// SIMATIC S7-200 project (STEP 7-Micro/WIN), CPU 224XP REL 02.01

SYMBOL_TABLE USER1
P0               M0.0
END_SYMBOL_TABLE

ORGANIZATION_BLOCK MAIN:OB1
TITLE=PROGRAM COMMENTS
BEGIN
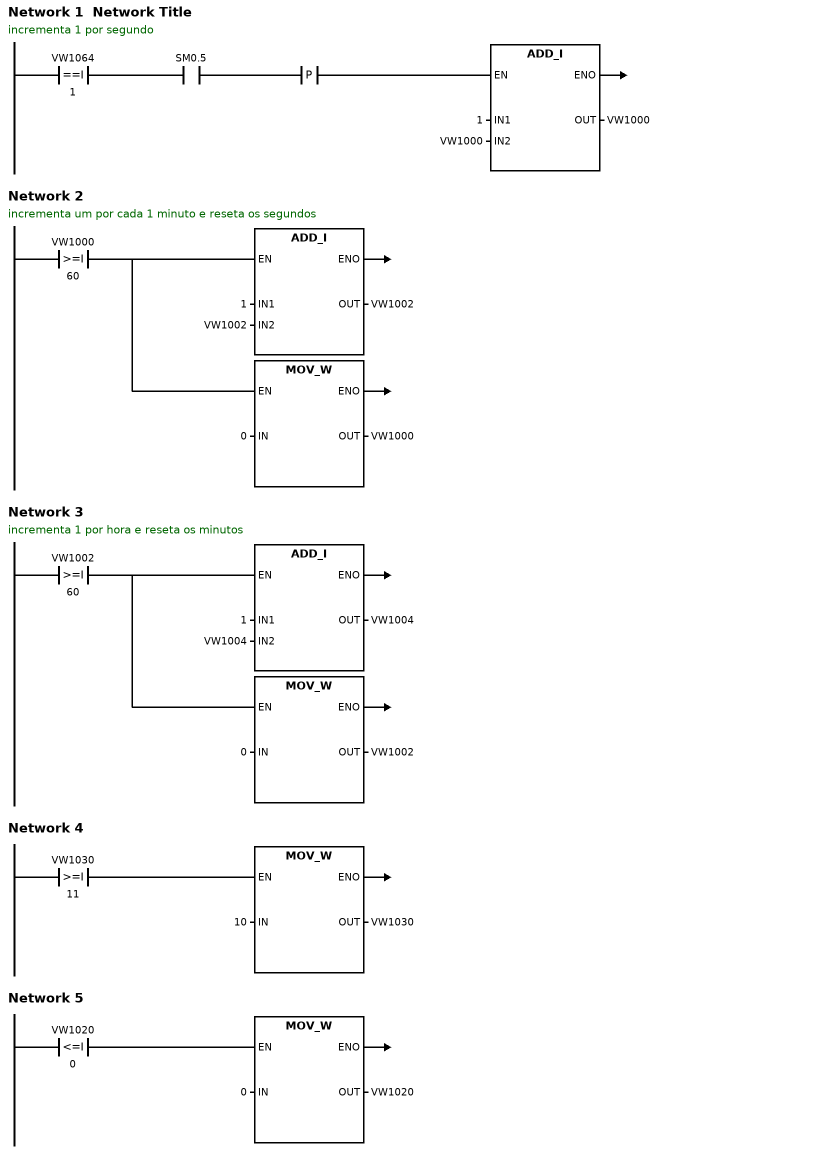
Network 1 // Network Title
// incrementa 1 por segundo
LDW=   VW1064, 1
A      SM0.5
EU
+I     1, VW1000
Network 2
// incrementa um por cada 1 minuto e reseta os segundos
LDW>=  VW1000, 60
+I     1, VW1002
MOVW   0, VW1000
Network 3
// incrementa 1 por hora e reseta os minutos
LDW>=  VW1002, 60
+I     1, VW1004
MOVW   0, VW1002
Network 4
LDW>=  VW1030, 11
MOVW   10, VW1030
Network 5
LDW<=  VW1020, 0
MOVW   0, VW1020
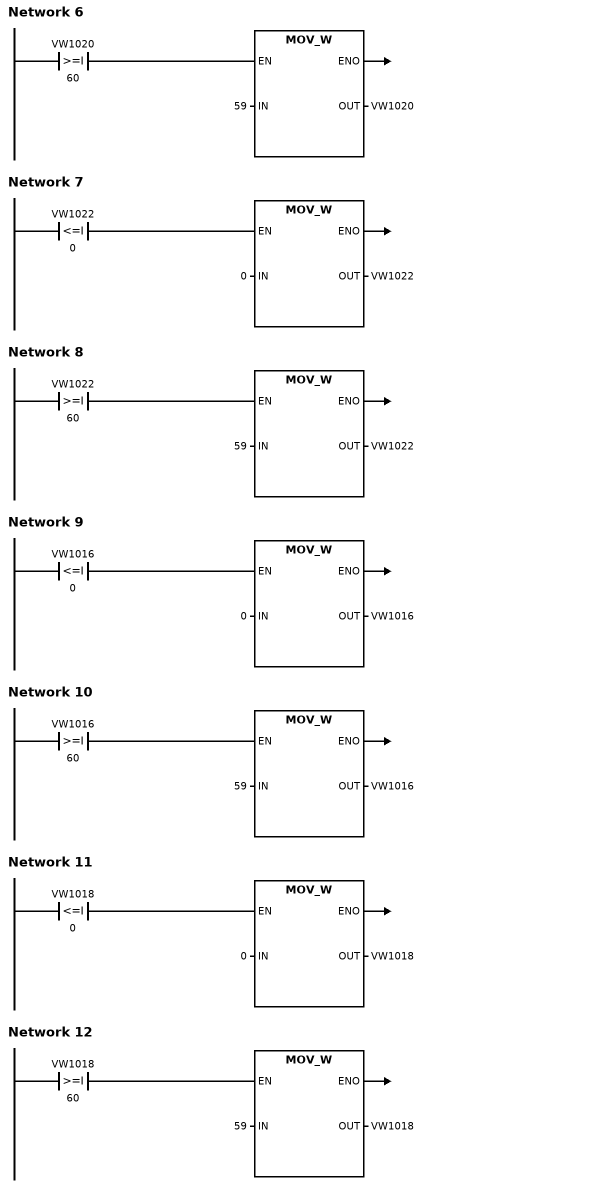
Network 6
LDW>=  VW1020, 60
MOVW   59, VW1020
Network 7
LDW<=  VW1022, 0
MOVW   0, VW1022
Network 8
LDW>=  VW1022, 60
MOVW   59, VW1022
Network 9
LDW<=  VW1016, 0
MOVW   0, VW1016
Network 10
LDW>=  VW1016, 60
MOVW   59, VW1016
Network 11
LDW<=  VW1018, 0
MOVW   0, VW1018
Network 12
LDW>=  VW1018, 60
MOVW   59, VW1018
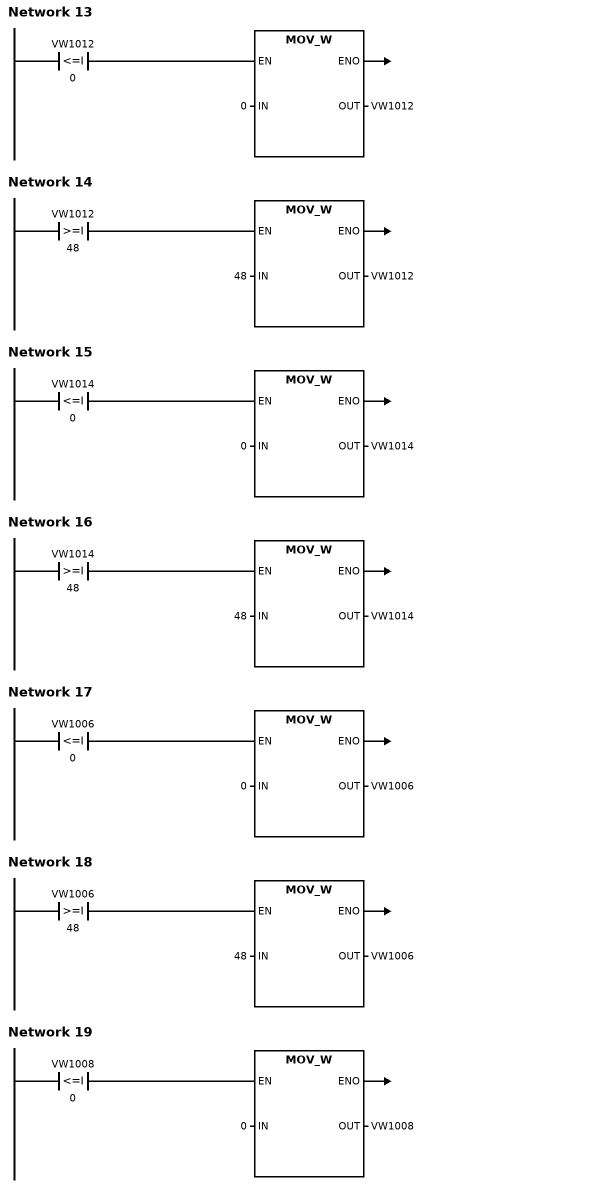
Network 13
LDW<=  VW1012, 0
MOVW   0, VW1012
Network 14
LDW>=  VW1012, 48
MOVW   48, VW1012
Network 15
LDW<=  VW1014, 0
MOVW   0, VW1014
Network 16
LDW>=  VW1014, 48
MOVW   48, VW1014
Network 17
LDW<=  VW1006, 0
MOVW   0, VW1006
Network 18
LDW>=  VW1006, 48
MOVW   48, VW1006
Network 19
LDW<=  VW1008, 0
MOVW   0, VW1008
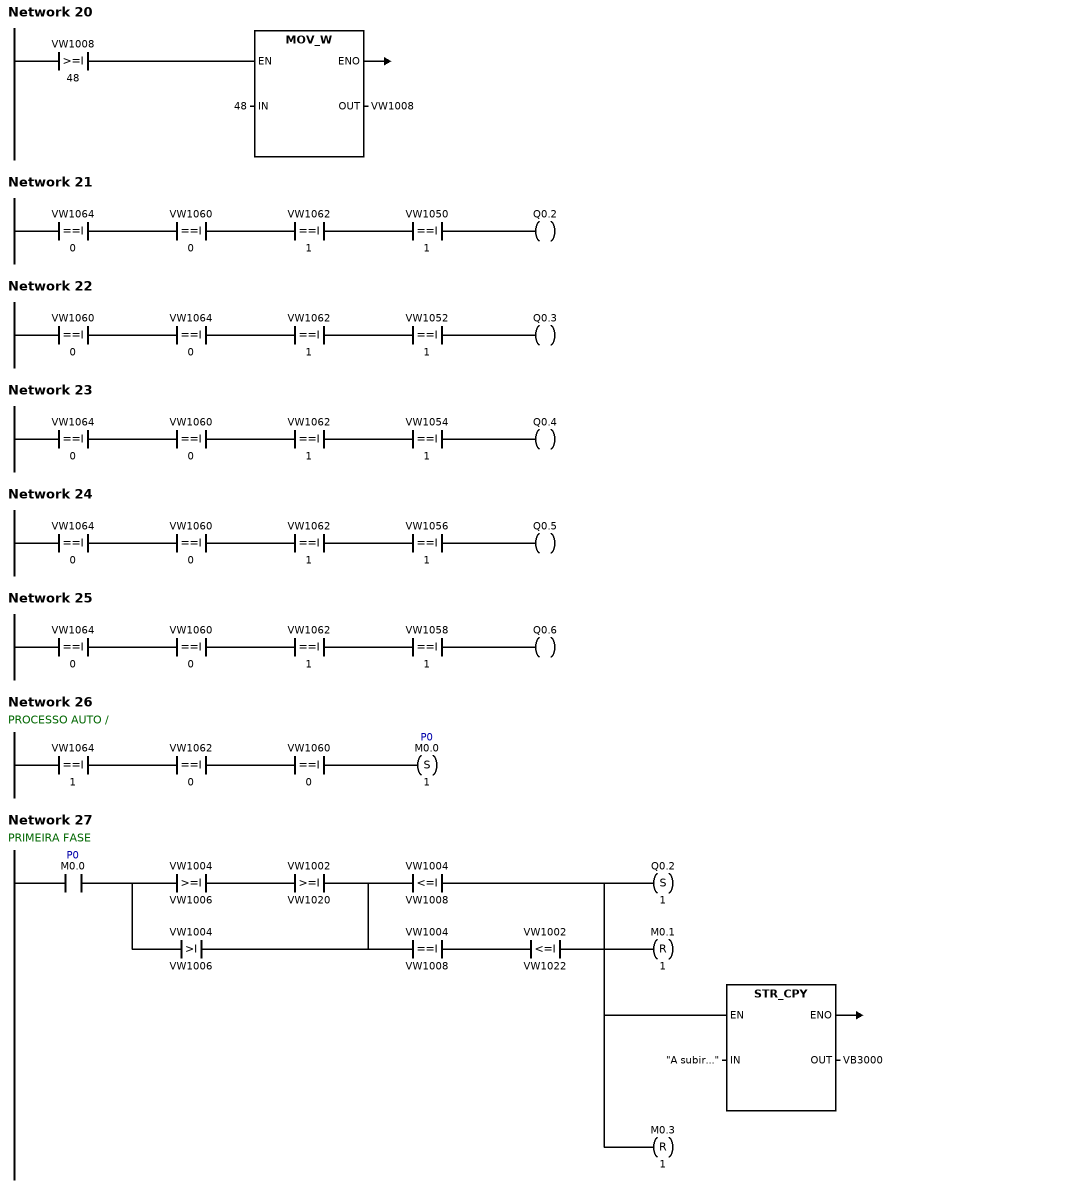
Network 20
LDW>=  VW1008, 48
MOVW   48, VW1008
Network 21
LDW=   VW1064, 0
AW=    VW1060, 0
AW=    VW1062, 1
AW=    VW1050, 1
=      Q0.2
Network 22
LDW=   VW1060, 0
AW=    VW1064, 0
AW=    VW1062, 1
AW=    VW1052, 1
=      Q0.3
Network 23
LDW=   VW1064, 0
AW=    VW1060, 0
AW=    VW1062, 1
AW=    VW1054, 1
=      Q0.4
Network 24
LDW=   VW1064, 0
AW=    VW1060, 0
AW=    VW1062, 1
AW=    VW1056, 1
=      Q0.5
Network 25
LDW=   VW1064, 0
AW=    VW1060, 0
AW=    VW1062, 1
AW=    VW1058, 1
=      Q0.6
Network 26
// PROCESSO AUTO
// 
LDW=   VW1064, 1
AW=    VW1062, 0
AW=    VW1060, 0
S      P0:M0.0, 1
Network 27
// PRIMEIRA FASE
LD     P0:M0.0
LDW>=  VW1004, VW1006
AW>=   VW1002, VW1020
OW>    VW1004, VW1006
ALD
LDW<=  VW1004, VW1008
LDW=   VW1004, VW1008
AW<=   VW1002, VW1022
OLD
ALD
S      Q0.2, 1
R      M0.1, 1
SCPY   "A subir...", VB3000
R      M0.3, 1
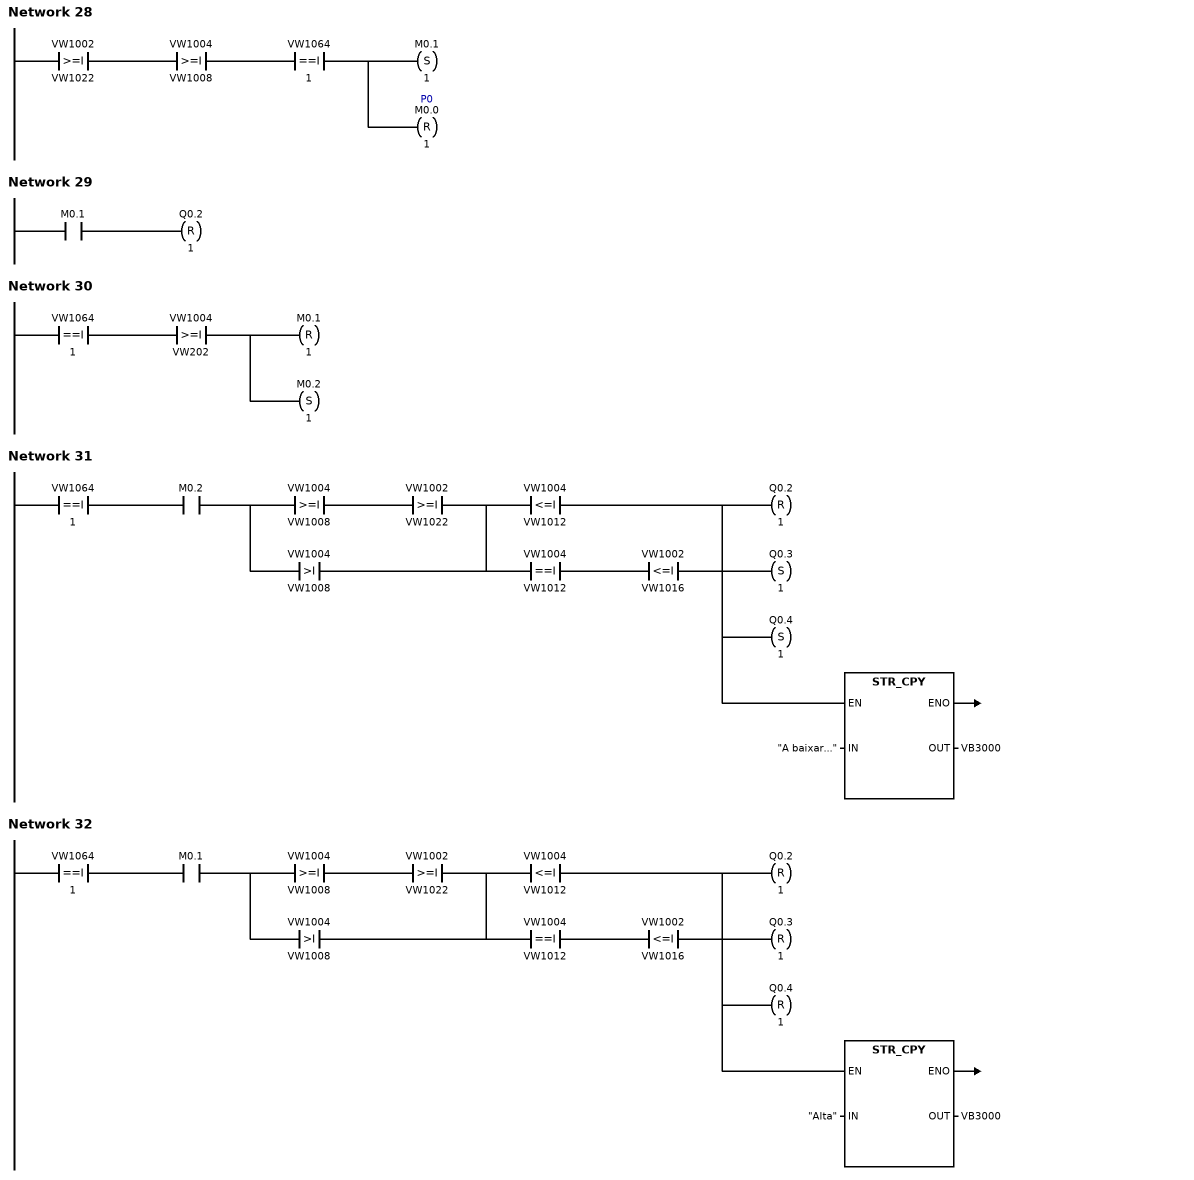
Network 28
LDW>=  VW1002, VW1022
AW>=   VW1004, VW1008
AW=    VW1064, 1
S      M0.1, 1
R      P0:M0.0, 1
Network 29
LD     M0.1
R      Q0.2, 1
Network 30
LDW=   VW1064, 1
AW>=   VW1004, VW202
R      M0.1, 1
S      M0.2, 1
Network 31
LDW=   VW1064, 1
A      M0.2
LDW>=  VW1004, VW1008
AW>=   VW1002, VW1022
OW>    VW1004, VW1008
ALD
LDW<=  VW1004, VW1012
LDW=   VW1004, VW1012
AW<=   VW1002, VW1016
OLD
ALD
R      Q0.2, 1
S      Q0.3, 1
S      Q0.4, 1
SCPY   "A baixar...", VB3000
Network 32
LDW=   VW1064, 1
A      M0.1
LDW>=  VW1004, VW1008
AW>=   VW1002, VW1022
OW>    VW1004, VW1008
ALD
LDW<=  VW1004, VW1012
LDW=   VW1004, VW1012
AW<=   VW1002, VW1016
OLD
ALD
R      Q0.2, 1
R      Q0.3, 1
R      Q0.4, 1
SCPY   "Alta", VB3000
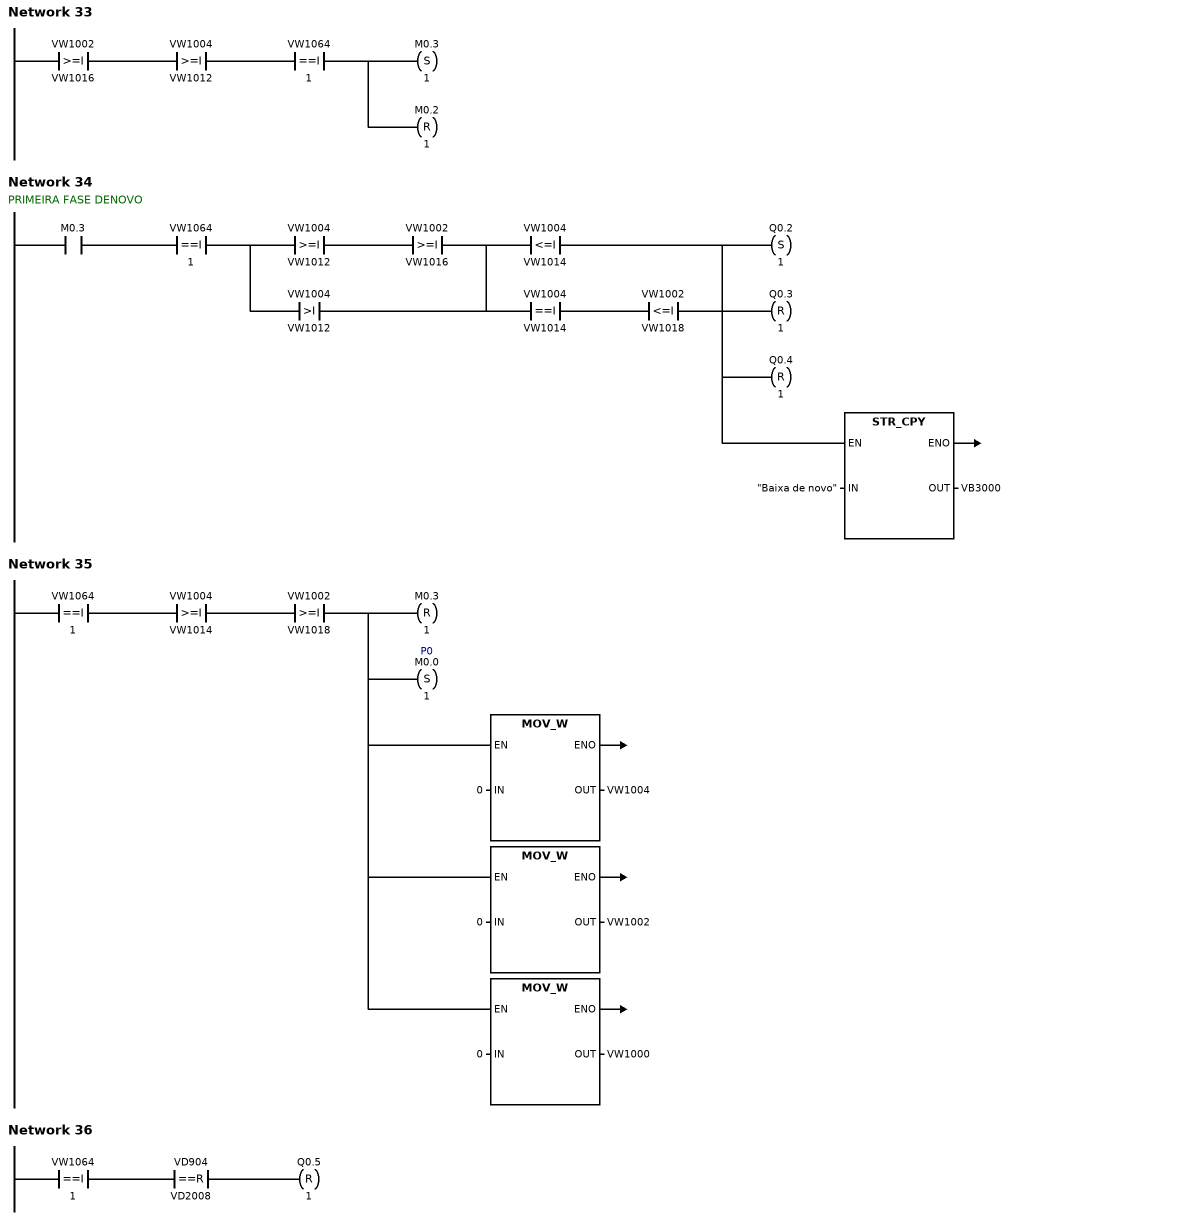
Network 33
LDW>=  VW1002, VW1016
AW>=   VW1004, VW1012
AW=    VW1064, 1
S      M0.3, 1
R      M0.2, 1
Network 34
// PRIMEIRA FASE DENOVO
LD     M0.3
AW=    VW1064, 1
LDW>=  VW1004, VW1012
AW>=   VW1002, VW1016
OW>    VW1004, VW1012
ALD
LDW<=  VW1004, VW1014
LDW=   VW1004, VW1014
AW<=   VW1002, VW1018
OLD
ALD
S      Q0.2, 1
R      Q0.3, 1
R      Q0.4, 1
SCPY   "Baixa de novo", VB3000
Network 35
LDW=   VW1064, 1
AW>=   VW1004, VW1014
AW>=   VW1002, VW1018
R      M0.3, 1
S      P0:M0.0, 1
MOVW   0, VW1004
MOVW   0, VW1002
MOVW   0, VW1000
Network 36
LDW=   VW1064, 1
AR=    VD904, VD2008
R      Q0.5, 1
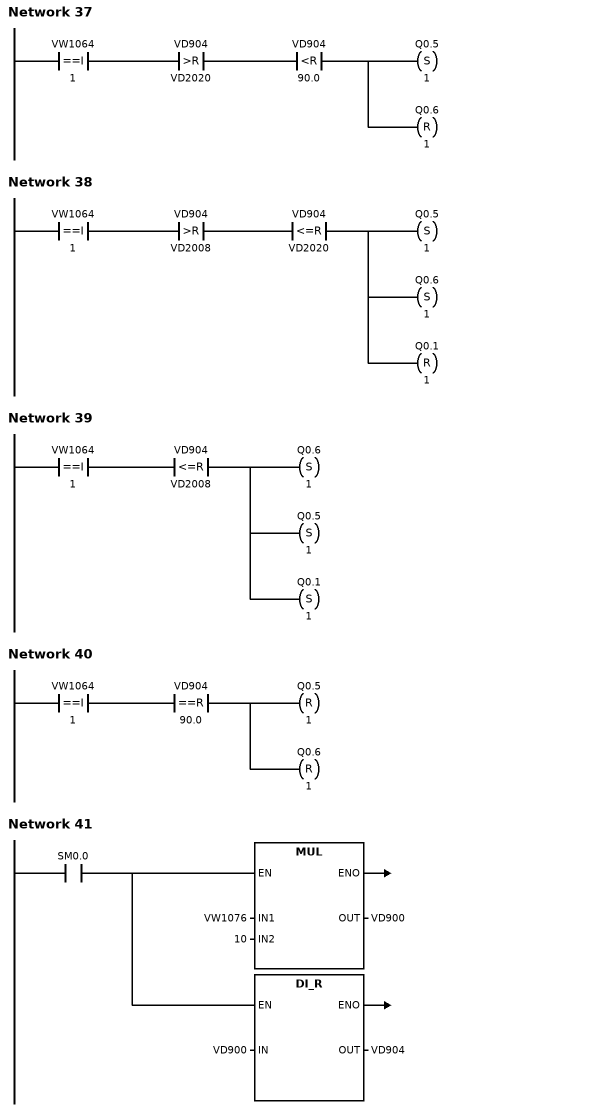
Network 37
LDW=   VW1064, 1
AR>    VD904, VD2020
AR<    VD904, 90.0
S      Q0.5, 1
R      Q0.6, 1
Network 38
LDW=   VW1064, 1
AR>    VD904, VD2008
AR<=   VD904, VD2020
S      Q0.5, 1
S      Q0.6, 1
R      Q0.1, 1
Network 39
LDW=   VW1064, 1
AR<=   VD904, VD2008
S      Q0.6, 1
S      Q0.5, 1
S      Q0.1, 1
Network 40
LDW=   VW1064, 1
AR=    VD904, 90.0
R      Q0.5, 1
R      Q0.6, 1
Network 41
LD     SM0.0
MOVW   VW1076, VW902
MUL    10, VD900
DTR    VD900, VD904
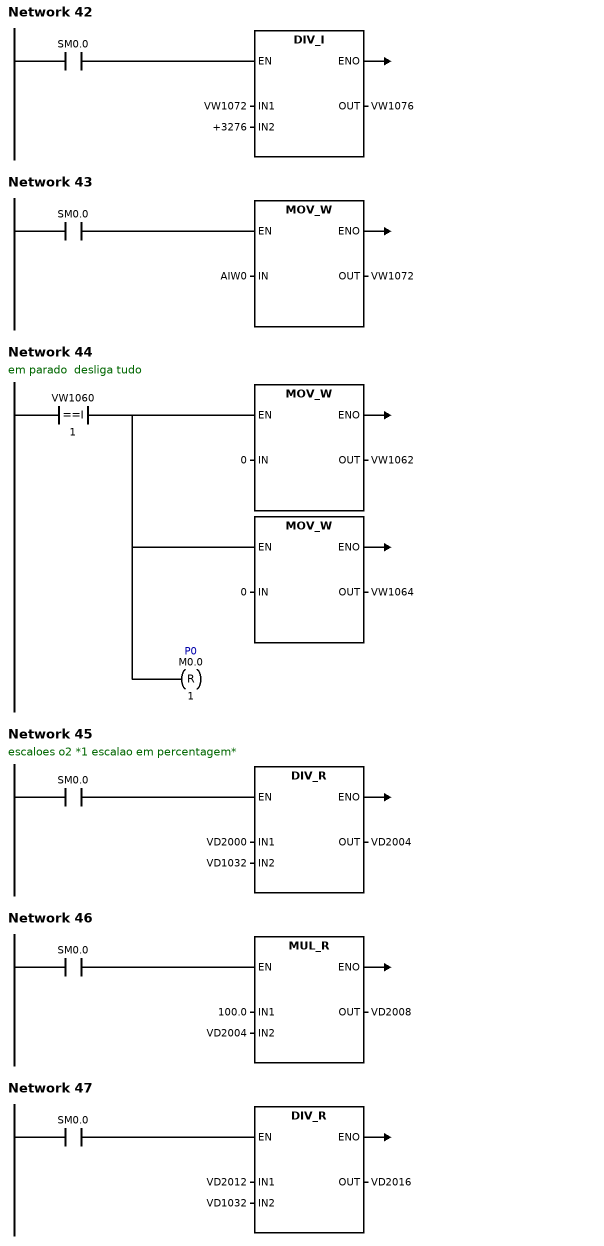
Network 42
LD     SM0.0
MOVW   VW1072, VW1076
/I     +3276, VW1076
Network 43
LD     SM0.0
MOVW   AIW0, VW1072
Network 44
// em parado  desliga tudo
LDW=   VW1060, 1
MOVW   0, VW1062
MOVW   0, VW1064
R      P0:M0.0, 1
Network 45
// escaloes o2 *1 escalao em percentagem*
LD     SM0.0
MOVR   VD2000, VD2004
/R     VD1032, VD2004
Network 46
LD     SM0.0
MOVR   100.0, VD2008
*R     VD2004, VD2008
Network 47
LD     SM0.0
MOVR   VD2012, VD2016
/R     VD1032, VD2016
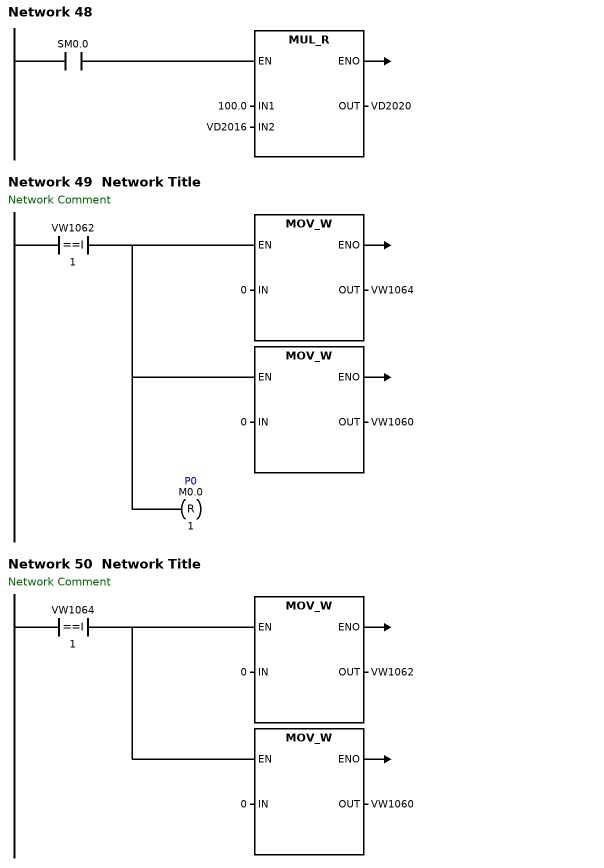
Network 48
LD     SM0.0
MOVR   100.0, VD2020
*R     VD2016, VD2020
Network 49 // Network Title
// Network Comment
LDW=   VW1062, 1
MOVW   0, VW1064
MOVW   0, VW1060
R      P0:M0.0, 1
Network 50 // Network Title
// Network Comment
LDW=   VW1064, 1
MOVW   0, VW1062
MOVW   0, VW1060
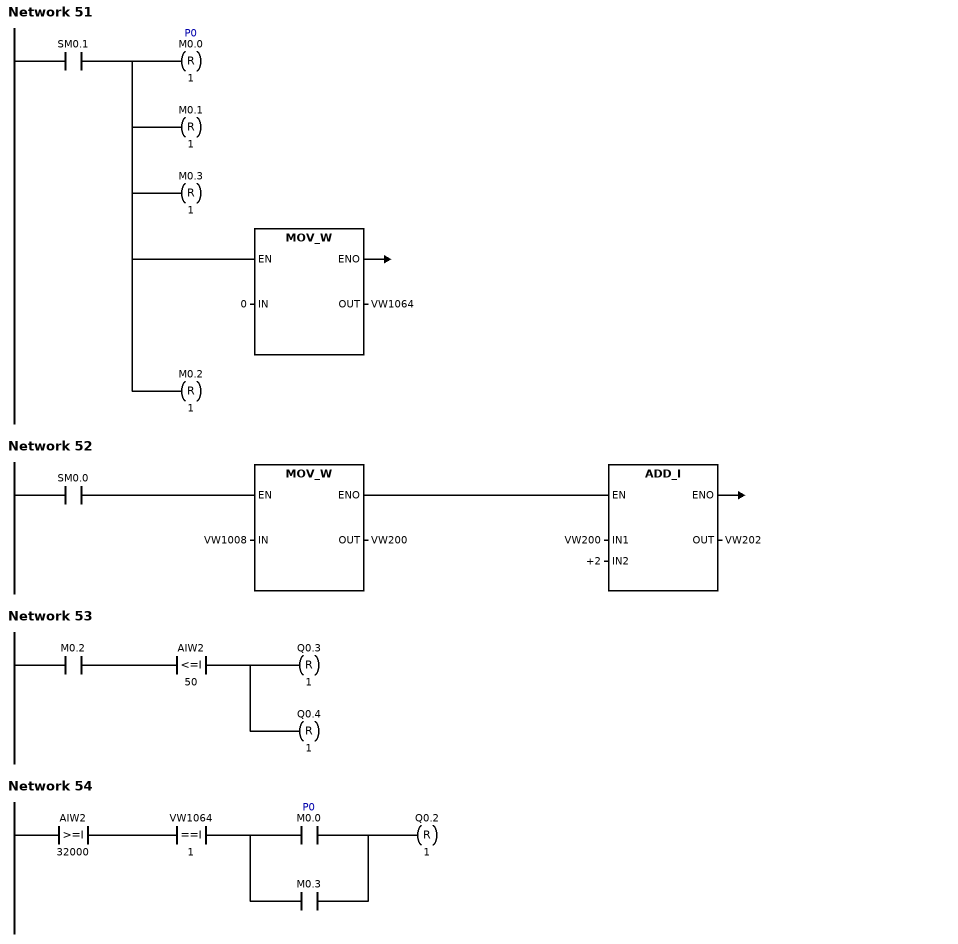
Network 51
LD     SM0.1
R      P0:M0.0, 1
R      M0.1, 1
R      M0.3, 1
MOVW   0, VW1064
R      M0.2, 1
Network 52
LD     SM0.0
MOVW   VW1008, VW200
AENO
MOVW   VW200, VW202
+I     +2, VW202
Network 53
LD     M0.2
AW<=   AIW2, 50
R      Q0.3, 1
R      Q0.4, 1
Network 54
LDW>=  AIW2, 32000
AW=    VW1064, 1
LD     P0:M0.0
O      M0.3
ALD
R      Q0.2, 1
END_ORGANIZATION_BLOCK

// SBR1: protected block, not included

// SBR2: protected block, not included

// (further data pages could not be read)
